INTERFACE I_Logger

METHOD LogCritical
VAR_INPUT
	Source	: I_TcSourceInfo;
    Message : T_MaxString;
END_VAR
END_METHOD

METHOD LogDebug
VAR_INPUT
	Source	: I_TcSourceInfo;
    Message : T_MaxString;
END_VAR
END_METHOD

METHOD LogError
VAR_INPUT
	Source	: I_TcSourceInfo;
    Message : T_MaxString;
END_VAR
END_METHOD

METHOD LogInfo
VAR_INPUT
	Source	: I_TcSourceInfo;
    Message : T_MaxString;
END_VAR
END_METHOD

METHOD LogWarning
VAR_INPUT
	Source	: I_TcSourceInfo;
    Message : T_MaxString;
END_VAR
END_METHOD

END_INTERFACE

(* stored: Version 1.1.0.1, ProductVersion 3.1.4024.15
   Itf I_Logger: Id {d6915353-f7c0-4c6f-b0da-5364769d4b0d}
   Method LogCritical: Id {6d6a42df-7810-48fa-9bac-d4259e669614}
   Method LogDebug: Id {0903a0cb-a44d-4638-86d5-a89b41aec2cb}
   Method LogError: Id {a1807b73-2133-4309-aa8e-36f133cadc56}
   Method LogInfo: Id {488d2f10-6234-4a74-9ecc-a8b29153f3c1}
   Method LogWarning: Id {85177536-4212-41a4-b833-0df1ae72a337} *)
